// TIA Portal V19 export
FUNCTION "FC_WORK_TO_POS" : Void   // FC54, STL
TITLE = Arbeitsdaten zurückschreiben
{ S7_Optimized_Access := 'FALSE' }
AUTHOR : MS
// Überträgt die Positionsdaten nach der Bearbeitung wieder in den Positions-DB
// stored: AutoNumber false
   VAR_INPUT
      Akt_Pos : USInt;   // Position die geladen wird
   END_VAR
BEGIN

NETWORK
TITLE = Move Dat
// von Feld[0] -- > [akt_pos]
      CALL  MOVE
      ( IN  := "DB_POS".POS[0],
        OUT := "DB_POS".POS[#Akt_Pos]
      );

END_FUNCTION
